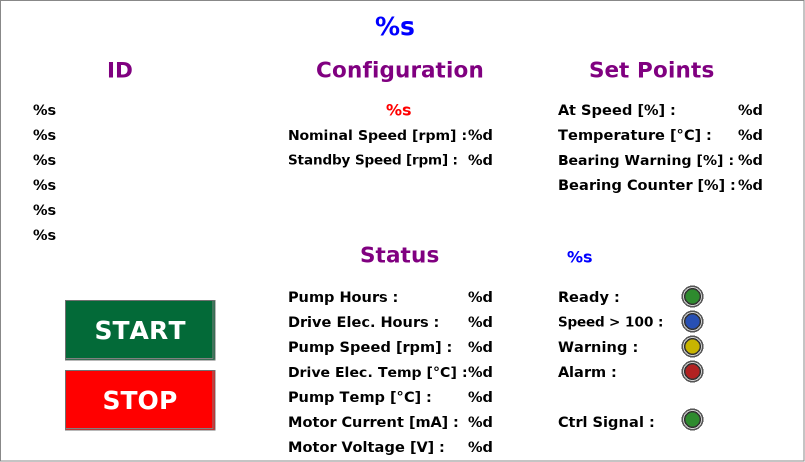
VISUALIZATION GUI_TEMPLATE_ATH2303M  // 805x462
VAR_IN_OUT
	m_Instance:	FB_CRYO_PUMP_ATH2303M;
	m_bEnable:	BOOL;	// Flag to start/stop the pump
END_VAR
    Rectangle (45,55 150x30), "ID"
    Rectangle (310,55 180x30), "Configuration"
    Rectangle (325,240 150x30), "Status"
    Lamp1 (680,284 25x25), tooltip "OK for Process, i.e. speed ≥ nominal speed", variable: m_Instance.stat.bReady, style: Lamp-Lamp1-Green
    Lamp1 (680,309 25x25), tooltip "pump speed > 100 rpm", variable: m_Instance.stat.bSpeed100, style: Lamp-Lamp1-Blue
    Lamp1 (680,334 25x25), tooltip "presence of a warning", variable: m_Instance.stat.bWarning, style: Lamp-Lamp1-Yellow
    Lamp1 (680,359 25x25), tooltip "presence of an alarm", variable: m_Instance.stat.bAlarm, style: Lamp-Lamp1-Red
    Rectangle (555,282 110x30), "Ready :"
    Rectangle (555,307 110x30), "Speed > 100 :"
    Rectangle (555,332 110x30), "Warning :"
    Rectangle (555,357 110x30), "Alarm :"
    Rectangle (30,145 240x30), "%s", text variable: m_Instance.stat.sVer1
    Rectangle (30,170 240x30), "%s", text variable: m_Instance.stat.sVer2
    Rectangle (30,195 240x30), "%s", text variable: m_Instance.stat.sVer3
    Rectangle (30,220 240x30), "%s", text variable: m_Instance.stat.sVer4
    Rectangle (285,120 180x30), "Nominal Speed [rpm] :"
    Rectangle (285,145 180x30), "Standby Speed [rpm] :"
    Rectangle (285,282 180x30), "Pump Hours :"
    Rectangle (285,307 180x30), "Drive Elec. Hours :"
    Rectangle (577,55 150x30), "Set Points"
    Rectangle (555,95 180x30), "At Speed [%] :"
    Rectangle (555,120 180x30), "Temperature [°C] :"
    Rectangle (555,145 180x30), "Bearing Warning [%] :"
    Rectangle (555,170 180x30), "Bearing Counter [%] :"
    Rectangle (735,95 70x30), "%d", text variable: m_Instance.stat.nSetPoint_AtSpeed
    Rectangle (735,120 70x30), "%d", text variable: m_Instance.stat.nSetPoint_Temp
    Rectangle (735,145 70x30), "%d", text variable: m_Instance.stat.nSetPoint_BearingWarn
    Rectangle (735,170 70x30), "%d", text variable: m_Instance.stat.nSetPoint_BearingCounter
    Rectangle (465,120 70x30), "%d", text variable: m_Instance.stat.nNominalSpeed
    Rectangle (465,145 70x30), "%d", text variable: m_Instance.stat.nStandbySpeed
    Rectangle (465,282 70x30), "%d", text variable: m_Instance.stat.nPumpHours
    Rectangle (465,307 70x30), "%d", text variable: m_Instance.stat.nElecHours
    Rectangle (285,332 180x30), "Pump Speed [rpm] :"
    Rectangle (465,332 70x30), "%d", text variable: m_Instance.stat.nPumpSpeed
    Rectangle (285,357 180x30), "Drive Elec. Temp [°C] :"
    Rectangle (465,357 70x30), "%d", text variable: m_Instance.stat.nElecTemp
    Rectangle (285,382 180x30), "Pump Temp [°C] :"
    Rectangle (465,382 70x30), "%d", text variable: m_Instance.stat.nPumpTemp
    Rectangle (285,407 180x30), "Motor Current [mA] :"
    Rectangle (465,407 70x30), "%d", text variable: m_Instance.stat.nMotorCurr
    Rectangle (285,432 180x30), "Motor Voltage [V] :"
    Rectangle (465,432 70x30), "%d", text variable: m_Instance.stat.nMotorVolt
    Rectangle (280,11 230x30), "%s", text variable: m_Instance.in_sName
    Rectangle (289,95 220x30), "%s", tooltip "Control Mode", text variable: m_Instance.stat.sCtrlMode
    Rectangle (30,95 240x30), "%s", text variable: m_Instance.stat.sIDN
    Rectangle (30,120 240x30), "%s", text variable: m_Instance.stat.sRDI
    Button (65,300 150x60), "START"
        OnMouseClick: execute { m_bEnable := TRUE; }
    Button (65,370 150x60), "STOP"
        OnMouseClick: execute { m_bEnable := FALSE; }
    Lamp1 (680,407 25x25), tooltip "If ON, control output signal is active.", variable: m_Instance.q_bStart, style: Lamp-Lamp1-Green
    Rectangle (555,407 110x30), "Ctrl Signal :"
    Rectangle (457,242 246x30), "%s", tooltip "Control Mode", text variable: m_Instance.stat.sPumpState
END_VISUALIZATION

(* stored: Version 1.1.0.1, ProductVersion 3.1.4024.12
   Visu GUI_TEMPLATE_ATH2303M: Id {96e9043d-3020-4847-9ef5-0a2e76d1852c} *)
